Universal Robots PolyScope program: circle.urp

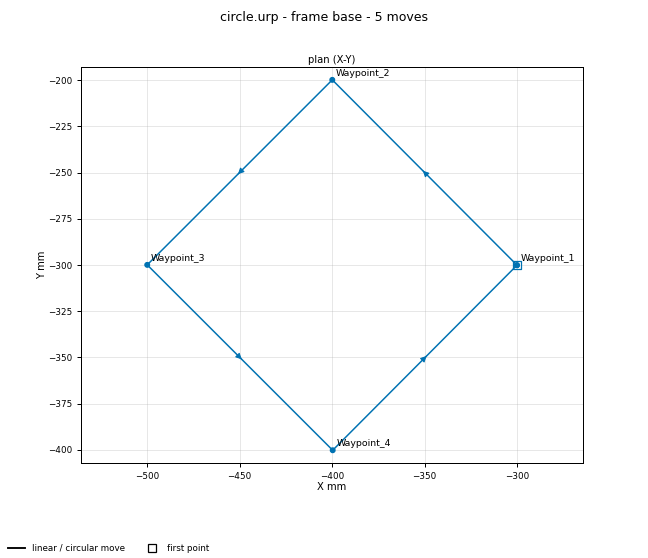
[picture p0: tool path of circle.urp in frame base, 5 of 5 moves have a stored position in this frame; points joined in program order, loops and branches not executed]
ProgramRoot directory=/home/ur/ursim-1.5/programs; kinematics=(a=[0, -0.425, -0.39243, 0, 0, 0], d=[0.0892, 0, 0, 0.109, 0.093, 0.082], alpha=[1.5708, 0, 0, 1.5708, -1.5708, 0], deltaTheta=[0, 0, 0, 0, 0, 0], status=notInitialized); name=circle; programVersion=(project__name=PolyScope, major__version=1, minor__version=5, svn__revision=7849, build__date=Feb 06 2012, 15:16:46); robotEnvironmentFileName=default
  MainProgram cartesianAcceleration=1.2; cartesianSpeed=0.25; jointAcceleration=1.3962634015954636; jointSpeed=1.0471975511965976; moveAsFastAsPossible=true; sharedProcessMoveBlendRadius=0.025; featureReference=(installationNameReference=Base); motionType=JOINT_SPACE
    Move cartesianAcceleration=1.2; cartesianSpeed=0.25; jointAcceleration=1.3962634015954636; jointSpeed=1.0471975511965976; moveAsFastAsPossible=true; sharedProcessMoveBlendRadius=0.025; featureReference=(installationNameReference=Base); motionType=PROCESS_MOVE
      Waypoint blendRadius=0.0; cartesianAcceleration=1.2; cartesianSpeed=0.25; jointAcceleration=1.3962634015954636; jointSpeed=1.0471975511965976; nextMotionTime=2.0; useSharedBlendParameter=true; useSharedParameters=true; position=TCP in base x=-300.031 y=-300.068 z=100.037 mm, rx=-2.6958 ry=1.6053 rz=-0.0366 rad; joints [29.907, -77.52, 132.345, -143.983, 271.058, 181.446] deg; positionType=FIXED_POSITION; waypointPoseInFeatureCoordinates=(pos=(x=-0.3000311766275814, y=-0.30006806343793485, z=0.100036731612092), rot=(x=-2.6958266290097836, y=1.6053174771728282, z=-0.03656568316875425)); name=Waypoint_1
      CircleMove insertableAsSuppressedNode=true; description=<html>Un movimento circolare viene effettuato con due punti percorso. Il primo specifica un punto sull'arco di circonferenza, mentre il secondo rappresenta l'endpoint del movimento.</html>; name=CircleMove
        Waypoint blendRadius=0.05; cartesianAcceleration=1.2; cartesianSpeed=0.25; jointAcceleration=1.3962634015954636; jointSpeed=1.0471975511965976; nextMotionTime=2.0; stoppoint=true; useSharedBlendParameter=true; useSharedParameters=true; position=TCP in base x=-399.919 y=-199.851 z=99.988 mm, rx=-2.6948 ry=1.6068 rz=-0.0376 rad; joints [12.294, -75.09, 128.737, -142.493, 270.778, 163.898] deg; positionType=FIXED_POSITION; waypointPoseInFeatureCoordinates=(pos=(x=-0.3999194397398224, y=-0.1998511134800707, z=0.0999881565281523), rot=(x=-2.6948434436189417, y=1.6068162558525159, z=-0.03760780910912858)); name=Waypoint_2
        Waypoint blendRadius=0.05; cartesianAcceleration=1.2; cartesianSpeed=0.25; jointAcceleration=1.3962634015954636; jointSpeed=1.0471975511965976; nextMotionTime=2.0; stoppoint=true; useSharedBlendParameter=true; useSharedParameters=true; position=TCP in base x=-500.001 y=-299.908 z=99.978 mm, rx=-2.6951 ry=1.6061 rz=-0.0381 rad; joints [20.048, -61.271, 106.422, -134.094, 270.933, 171.623] deg; positionType=FIXED_POSITION; waypointPoseInFeatureCoordinates=(pos=(x=-0.5000012332166232, y=-0.2999082119074865, z=0.09997841760005603), rot=(x=-2.6950961061374907, y=1.6060773985237407, z=-0.03807545791718738)); name=Waypoint_3
      CircleMove insertableAsSuppressedNode=true; description=<html>Un movimento circolare viene effettuato con due punti percorso. Il primo specifica un punto sull'arco di circonferenza, mentre il secondo rappresenta l'endpoint del movimento.</html>; name=CircleMove
        Waypoint blendRadius=0.05; cartesianAcceleration=1.2; cartesianSpeed=0.25; jointAcceleration=1.3962634015954636; jointSpeed=1.0471975511965976; nextMotionTime=2.0; stoppoint=true; useSharedBlendParameter=true; useSharedParameters=true; position=TCP in base x=-399.692 y=-400.168 z=100.021 mm, rx=-2.6955 ry=1.6054 rz=-0.0383 rad; joints [33.75, -63.034, 109.541, -135.7, 271.164, 185.296] deg; positionType=FIXED_POSITION; waypointPoseInFeatureCoordinates=(pos=(x=-0.3996917314569661, y=-0.40016765793989867, z=0.10002074179221776), rot=(x=-2.6955428879660936, y=1.6053790838185067, z=-0.0382724407140308)); name=Waypoint_4
        Waypoint blendRadius=0.0; cartesianAcceleration=1.2; cartesianSpeed=0.25; jointAcceleration=1.3962634015954636; jointSpeed=1.0471975511965976; nextMotionTime=2.0; useSharedBlendParameter=true; useSharedParameters=true; position=TCP in base x=-300.055 y=-300.122 z=100.089 mm, rx=-2.6964 ry=1.6051 rz=-0.0368 rad; joints [29.909, -77.521, 132.34, -143.988, 271.074, 181.43] deg; positionType=FIXED_POSITION; waypointPoseInFeatureCoordinates=(pos=(x=-0.3000545661892398, y=-0.3001220479458041, z=0.10008900534890271), rot=(x=-2.696351508548074, y=1.6050677887877463, z=-0.036766003277165)); name=Waypoint_5
